FUNCTION_BLOCK FB_HE_SATT_FilterConstantThickness EXTENDS FB_HE_SATT_Filter IMPLEMENTS I_HE_SATT_FilterConstantThickness
VAR
    fThickness : LREAL;
END_VAR


METHOD FB_Init: BOOL
VAR_INPUT
    bInitRetains: BOOL; // TRUE: the retain variables are initialized (reset warm / reset cold)
    bInCopyCode: BOOL;  // TRUE: the instance will be copied to the copy code afterward (online change)   
    
    iHolder : I_HE_SATT_FilterHolder;
    fDefaultLength : LREAL;
    eDefaultMaterial : E_HE_SATT_FilterMaterial;
    eDefaultStatus : E_HE_SATT_FilterStatus;
    fDefaultThickness : LREAL;
END_VAR

THIS^.iHolder := iHolder;
THIS^.fLength := fDefaultLength;
THIS^.eMaterial := eDefaultMaterial;
THIS^.eStatus := eDefaultStatus;
THIS^.fThickness := fDefaultThickness;
END_METHOD


PROPERTY Thickness : LREAL
GET

Thickness := THIS^.fThickness;
END_GET
SET

THIS^.fThickness := Thickness;
END_SET
END_PROPERTY

END_FUNCTION_BLOCK

(* stored: Version 1.1.0.1
   POU FB_HE_SATT_FilterConstantThickness: Id {27eb9296-9818-4e4c-9c08-09c6b3b98b53}, SpecialFunc None
   Method FB_Init: Id {d5a8aecc-ba29-4911-9e4d-7d067aaef986}
   Property Thickness: Id {6dd1d3c7-656a-4c9b-b053-808645967324}
   Get Get: Id {3646f10f-d718-4286-aa4e-965c5869e721}
   Set Set: Id {d6929622-549a-42d6-a755-38791c9f4524} *)
